Fanuc TP program (LS listing): FOLGE020.LS

/PROG  FOLGE020
/ATTR
OWNER		= AUROM;
COMMENT		= "VW336";
PROG_SIZE	= 5438;
CREATE		= DATE 96-03-31  TIME 20:16:44;
MODIFIED	= DATE 23-07-08  TIME 16:53:20;
FILE_NAME	= FOLGE020;
VERSION		= 0;
LINE_COUNT	= 30;
MEMORY_SIZE	= 8818;
PROTECT		= READ_WRITE;
TCD:  STACK_SIZE	= 500,
      TASK_PRIORITY	= 50,
      TIME_SLICE	= 0,
      BUSY_LAMP_OFF	= 0,
      ABORT_REQUEST	= 0,
      PAUSE_REQUEST	= 0;
DEFAULT_GROUP	= 1,1,1,1,*;
CONTROL_CODE	= 00000000 00000000;
/APPL
/MN
   1:  UTOOL_NUM=1 ;
   2:  UFRAME_NUM=0 ;
   3:  PAYLOAD[1] ;
   4:J P[1] 10% CNT0 ACC100 TB   0.00sec,P-SPS    ;
      1:  IF (DO[12]),CALL MAKRO998 ;
      2:  DO[15]=ON ;
      3:  DO[16]=ON ;
      4:  CALL MAKRO000    ;
      5:  WAIT (DI[9])    ;
       ------ ;
   5:  !Fresado Estacionario ;
   6:J P[2] 100% CNT0 ACC100 TB   0.00sec,P-SPS    ;
      1:  TC_ONLINE (ON) ;
      2:  DO[23]=OFF ;
      3:  TIMER[1]=RESET ;
      4:  TIMER[1]=START ;
      5:  CALL MAKRO050    ;
      6:  !Lib. de Herramientas ;
      7:  DO[80]=ON ;
      8:  DO[78]=OFF ;
      9:  DO[76]=ON ;
     10:  DO[74]=OFF ;
     11:  !Lib. de Anticolisiones ;
     12:  DO[41]=ON ;
     13:  DO[42]=ON ;
     14:  !Apagar Posicion Base ;
     15:  DO[15]=OFF ;
     16:  !Garra a Base si no hay pieza ;
     17:  WAIT (M[2])    ;
     18:  F[1]=(ON) ;
     19:  F[2]=(ON) ;
     20:  F[3]=(ON) ;
     21:  IF (M[2]),CALL MAKRO342 ;
     22:  CALL MAKRO340    ;
     23:  WAIT (M[31] AND M[33] AND M[35])    ;
     24:  !Fresado SZ1 ;
     25:  F[298]=(OFF) ;
     26:  CALL VW_USER(Basic1,EZSP,Nr1 Service,ProgNr=31, , ,S-Punkt=31, ,EIN/AUS=ON) ;
     27:  WAIT    .10(sec) ;
     28:  F[79]=((DI[786] AND !DI[788]) OR (!DI[788] AND DI[130])) ;
     29:  F[78]=(DI[788] AND !F[79]) ;
     30:  GO[2]=(R[197]+5) ;
     31:  IF (F[78] OR F[79]),CALL MAKRO085 ;
     32:  IF (F[78] OR F[79]),CALL MAKRO084 ;
     33:  WAIT (M[96])    ;
     34:  WAIT (DI[23])    ;
     35:  DO[23]=ON ;
     36:  TC_ONLINE (M[2] AND M[30] AND M[31] AND M[33] AND M[35] AND M[95] AND M[96]) ;
       ------ ;
   7:  !Llamar a UP021 ;
   8:  !Tomar De ST1180 ;
   9:J P[3] 100% CNT0 ACC100 TB    .10sec,P-SPS    ;
      1:  TC_ONLINE (ON) ;
      2:  DO[23]=OFF ;
      3:  WAIT (DI[23])    ;
      4:  DO[23]=ON ;
      5:  TC_ONLINE (M[2] AND M[30] AND M[31] AND M[33] AND M[35] AND M[95] AND M[96]) ;
       ------ ;
  10:  CALL UP021    ;
  11:  UFRAME_NUM=0 ;
  12:  UTOOL_NUM=1 ;
  13:  !Llamar a UP022 ;
  14:  !Soldadura Estacionaria ;
  15:J P[4] 100% CNT0 ACC100 TB    .10sec,P-SPS    ;
      1:  TC_ONLINE (ON) ;
      2:  DO[23]=OFF ;
      3:  WAIT (DI[23])    ;
      4:  DO[23]=ON ;
      5:  TC_ONLINE (M[1] AND M[30] AND M[32] AND M[34] AND M[35] AND M[95] AND M[96]) ;
       ------ ;
  16:  CALL UP022    ;
  17:  UFRAME_NUM=0 ;
  18:  UTOOL_NUM=1 ;
  19:  ! En Area de Mantenimiento ;
  20:  ! Llamar a UP023 ;
  21:  ! Depositar en Banda 1300 ;
  22:J P[5] 100% CNT0 ACC100 TB    .10sec,P-SPS    ;
      1:  TC_ONLINE (ON) ;
      2:  DO[23]=OFF ;
      3:  LBL[1] ;
      4:  DO[18]=(ON) ;
      5:  WAIT ((DI[76] AND !DI[62] AND DI[61] AND !DI[18]) OR DI[19])    ;
      6:  IF (DI[19]),JMP LBL[3] ;
      7:  IF (DI[76]),JMP LBL[2] ;
      8:  LBL[3] ;
      9:  IF (F[78] OR F[79]),CALL MAKRO084 ;
     10:  CALL MAKRO089    ;
     11:  DO[17]=(ON) ;
     12:  GO[19]=(11) ;
     13:  F[281]=(ON) ;
     14:  WAIT (DI[17])    ;
     15:  F[64]=(ON) ;
     16:  F[65]=(OFF) ;
     17:  F[66]=(OFF) ;
     18:  F[67]=(OFF) ;
     19:  LBL[4] ;
     20:  IF (DI[132] AND !DI[133] AND !DI[134] AND !DI[135] AND DI[17]),CALL MAKRO081 ;
     21:  IF (F[85]),JMP LBL[4] ;
     22:  CALL VW_USER(Basic1,EZSP,Nr1 Service,ProgNr=31, , ,S-Punkt=31, ,EIN/AUS=ON) ;
     23:  F[79]=((!DI[788] AND DI[130]) OR (DI[786] AND !DI[788])) ;
     24:  F[78]=(DI[788] AND !F[79]) ;
     25:  GO[2]=(R[197]+5) ;
     26:  IF (F[78] OR F[79]),CALL MAKRO085 ;
     27:  IF (F[78] OR F[79]),CALL MAKRO084 ;
     28:  WAIT (M[96] AND !DI[132])    ;
     29:  DO[17]=(OFF) ;
     30:  GO[19]=(0) ;
     31:  WAIT (!DI[19])    ;
     32:  JMP LBL[1] ;
     33:  LBL[2] ;
     34:  DO[18]=(OFF) ;
     35:  F[281]=(OFF) ;
     36:  WAIT (DI[23])    ;
     37:  DO[23]=ON ;
     38:  TC_ONLINE (M[1] AND M[30] AND M[32] AND M[34] AND M[35] AND M[95] AND M[96]) ;
       ------ ;
  23:  CALL UP023    ;
  24:  UFRAME_NUM=0 ;
  25:  UTOOL_NUM=1 ;
  26:  !Fresado Estacionario ;
  27:J P[6] 100% CNT0 ACC100 TB    .10sec,P-SPS    ;
      1:  TC_ONLINE (ON) ;
      2:  DO[23]=OFF ;
      3:  !Fresado SZ1 ;
      4:  CALL VW_USER(Basic1,EZSP,Nr1 Service,ProgNr=31, , ,S-Punkt=31, ,EIN/AUS=ON) ;
      5:  WAIT    .10(sec) ;
      6:  F[79]=((DI[786] AND !DI[788]) OR (!DI[788] AND DI[130])) ;
      7:  F[78]=(DI[788] AND !F[79]) ;
      8:  GO[2]=(R[197]+5) ;
      9:  IF (F[78] OR F[79]),CALL MAKRO085 ;
     10:  IF (F[78] OR F[79]),CALL MAKRO084 ;
     11:  WAIT (M[96])    ;
     12:  WAIT (DI[23])    ;
     13:  DO[23]=ON ;
     14:  TC_ONLINE (M[2] AND M[30] AND M[31] AND M[33] AND M[35] AND M[95] AND M[96]) ;
       ------ ;
  28:  !Fin de trabajo total ;
  29:J P[7] 100% CNT0 ACC100 TB    0.00sec,P-SPS    ;
      1:  TC_ONLINE (ON) ;
      2:  DO[23]=OFF ;
      3:  CALL MAKRO015    ;
      4:  WAIT (DI[23])    ;
      5:  DO[23]=ON ;
      6:  TC_ONLINE (M[2] AND M[30] AND M[31] AND M[33] AND M[35] AND M[95] AND M[96]) ;
       ------ ;
  30:J P[8] 100% CNT0 ACC100 TB   0.00sec,P-SPS    ;
      1:  TC_ONLINE (ON) ;
      2:  DO[14]=ON ;
      3:  DO[15]=ON ;
      4:  TIMER[1]=STOP ;
      5:  TIMER[2]=(TIMER[1]) ;
      6:  TIMER[2]=STOP ;
       ------ ;
/POS
P[1]{
   GP1:
	UF : 0, UT : 1,		CONFIG : 'F U T, 0, 0, 0',
	X =   124.280  mm,	Y =    20.861  mm,	Z =  2168.892  mm,
	W =  -108.055 deg,	P =   -84.588 deg,	R =    68.064 deg
   GP2:
	UF : 0, UT : 1,
	J1=   168.000  mm
   GP3:
	UF : 0, UT : 1,
	J1=     0.000  mm
   GP4:
	UF : 0, UT : 1,
	J1=     0.000  mm
};
P[2]{
   GP1:
	UF : 0, UT : 1,		CONFIG : 'F U T, 0, 0, 0',
	X =   124.280  mm,	Y =    20.861  mm,	Z =  2168.892  mm,
	W =  -108.055 deg,	P =   -84.588 deg,	R =    68.064 deg
   GP2:
	UF : 0, UT : 1,
	J1=   168.000  mm
   GP3:
	UF : 0, UT : 1,
	J1=     0.000  mm
   GP4:
	UF : 0, UT : 1,
	J1=     0.000  mm
};
P[3]{
   GP1:
	UF : 0, UT : 1,		CONFIG : 'F U T, 0, 0, 0',
	X =   124.280  mm,	Y =    20.861  mm,	Z =  2168.892  mm,
	W =  -108.055 deg,	P =   -84.588 deg,	R =    68.064 deg
   GP2:
	UF : 0, UT : 1,
	J1=   168.000  mm
   GP3:
	UF : 0, UT : 1,
	J1=     0.000  mm
   GP4:
	UF : 0, UT : 1,
	J1=     0.000  mm
};
P[4]{
   GP1:
	UF : 0, UT : 1,		CONFIG : 'F U T, 0, 0, 0',
	X =   124.280  mm,	Y =    20.861  mm,	Z =  2168.892  mm,
	W =  -108.055 deg,	P =   -84.588 deg,	R =    68.064 deg
   GP2:
	UF : 0, UT : 1,
	J1=   168.000  mm
   GP3:
	UF : 0, UT : 1,
	J1=     0.000  mm
   GP4:
	UF : 0, UT : 1,
	J1=     0.000  mm
};
P[5]{
   GP1:
	UF : 0, UT : 1,		CONFIG : 'F U T, 0, 0, 0',
	X =   124.280  mm,	Y =    20.861  mm,	Z =  2168.892  mm,
	W =  -108.055 deg,	P =   -84.588 deg,	R =    68.064 deg
   GP2:
	UF : 0, UT : 1,
	J1=   168.000  mm
   GP3:
	UF : 0, UT : 1,
	J1=     0.000  mm
   GP4:
	UF : 0, UT : 1,
	J1=     0.000  mm
};
P[6]{
   GP1:
	UF : 0, UT : 1,		CONFIG : 'F U T, 0, 0, 0',
	X =   124.280  mm,	Y =    20.861  mm,	Z =  2168.892  mm,
	W =  -108.055 deg,	P =   -84.588 deg,	R =    68.064 deg
   GP2:
	UF : 0, UT : 1,
	J1=   168.000  mm
   GP3:
	UF : 0, UT : 1,
	J1=     0.000  mm
   GP4:
	UF : 0, UT : 1,
	J1=     0.000  mm
};
P[7]{
   GP1:
	UF : 0, UT : 1,		CONFIG : 'F U T, 0, 0, 0',
	X =   124.280  mm,	Y =    20.861  mm,	Z =  2168.892  mm,
	W =  -108.055 deg,	P =   -84.588 deg,	R =    68.064 deg
   GP2:
	UF : 0, UT : 1,
	J1=   168.000  mm
   GP3:
	UF : 0, UT : 1,
	J1=     0.000  mm
   GP4:
	UF : 0, UT : 1,
	J1=     0.000  mm
};
P[8]{
   GP1:
	UF : 0, UT : 1,		CONFIG : 'F U T, 0, 0, 0',
	X =   124.280  mm,	Y =    20.861  mm,	Z =  2168.892  mm,
	W =  -108.055 deg,	P =   -84.588 deg,	R =    68.064 deg
   GP2:
	UF : 0, UT : 1,
	J1=   168.000  mm
   GP3:
	UF : 0, UT : 1,
	J1=     0.000  mm
   GP4:
	UF : 0, UT : 1,
	J1=     0.000  mm
};
/END
